FUNCTION_BLOCK FB_BaseTest EXTENDS TcUnit.FB_TestSuite
VAR
	fbTest				: FB_Base;
END_VAR


T01_VariableBindingTest ();

METHOD PRIVATE T01_VariableBindingTest
VAR_INPUT
END_VAR

VAR
	bWynik: BOOL;
END_VAR
IF (TcUnit.TEST_ORDERED ('T01_VariableBindingTest')) THEN
	GVL.stCommonData.itfTime				:= GVL.fbMyTime;
	GVL.stCommonData.itfLocaciotn			:= GVL.fbMyLocation;
	GVL.stCommonData.itfLogger				:= GVL.fbLogger;
	
	bWynik		:= GVL_Variable.fbBasetest.LinkCommonData (stCommonData	:= GVL.stCommonData);
	
	AssertTrue (Condition := bWynik, Message := 'T01 - test utworezenia referencji');
	
	TcUnit.TEST_FINISHED ();
END_IF
END_METHOD

END_FUNCTION_BLOCK

(* stored: Version 1.1.0.1, ProductVersion 3.1.4024.15
   POU FB_BaseTest: Id {7ad8b220-f045-480c-8f86-96620e4491f8}, SpecialFunc None
   Method T01_VariableBindingTest: Id {015d9e92-fd3d-4e93-8815-35c0328a710d} *)
